Staubli VAL3: stop.pgx

program stop()
begin
  //$jogPage(true)
  //  title("")
  //  cls()
  //  call ListPop("EndOfProgram")
  //  resetMotion()
  libSave()
  bFinish=true
end
